SYSTEM PubSubTest
  (* Version 1.0, 2026-02-25, Administrateur *)
  APPLICATION PubSubTestApp
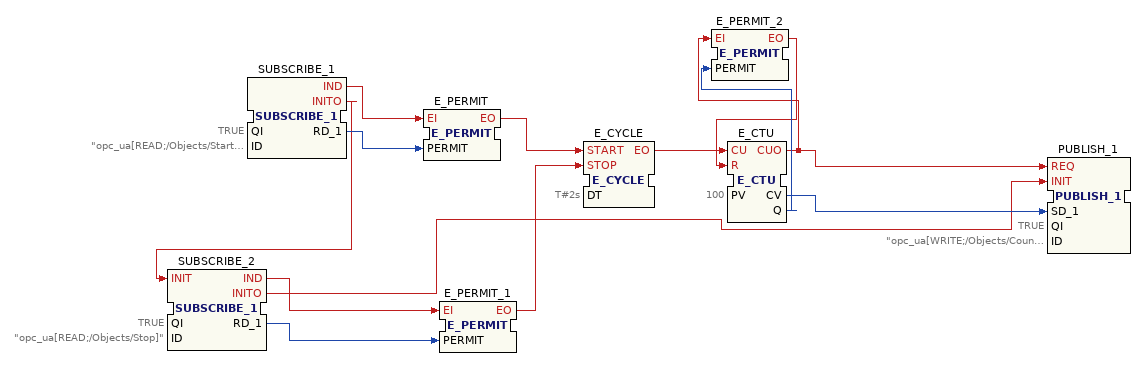
    FBS
      E_CYCLE : iec61499::events::E_CYCLE(DT := T#2s);
      E_CTU : iec61499::events::E_CTU(PV := 100);
      PUBLISH_1 : iec61499::net::PUBLISH_1(QI := TRUE, ID := "opc_ua[WRITE;/Objects/Counter]");
      SUBSCRIBE_1 : iec61499::net::SUBSCRIBE_1(QI := TRUE, ID := "opc_ua[READ;/Objects/Start]");
      E_PERMIT : iec61499::events::E_PERMIT;
      SUBSCRIBE_2 : iec61499::net::SUBSCRIBE_1(QI := TRUE, ID := "opc_ua[READ;/Objects/Stop]");
      E_PERMIT_1 : iec61499::events::E_PERMIT;
      E_PERMIT_2 : iec61499::events::E_PERMIT;
    END_FBS
    EVENT_CONNECTIONS
      E_CYCLE.EO TO E_CTU.CU;
      E_CTU.CUO TO PUBLISH_1.REQ;
      SUBSCRIBE_1.IND TO E_PERMIT.EI;
      E_PERMIT.EO TO E_CYCLE.START;
      E_PERMIT_1.EO TO E_CYCLE.STOP;
      SUBSCRIBE_2.IND TO E_PERMIT_1.EI;
      SUBSCRIBE_1.INITO TO SUBSCRIBE_2.INIT;
      SUBSCRIBE_2.INITO TO PUBLISH_1.INIT;
      E_CTU.CUO TO E_PERMIT_2.EI;
      E_PERMIT_2.EO TO E_CTU.R;
    END_CONNECTIONS
    DATA_CONNECTIONS
      E_CTU.CV TO PUBLISH_1.SD_1;
      SUBSCRIBE_1.RD_1 TO E_PERMIT.PERMIT;
      SUBSCRIBE_2.RD_1 TO E_PERMIT_1.PERMIT;
      E_CTU.Q TO E_PERMIT_2.PERMIT;
    END_CONNECTIONS
  END_APPLICATION
  DEVICE FORTE_PC : iec61499::system::FORTE_PC(MGR_ID := "localhost:61499" (* Device manager socket ID *))
    {SET_ATTRIBUTE(Profile, HOLOBLOC)}
    RESOURCE EMB_RES : iec61499::system::EMB_RES
      EVENT_CONNECTIONS
        START.WARM TO PubSubTestApp.SUBSCRIBE_1.INIT;
        START.COLD TO PubSubTestApp.SUBSCRIBE_1.INIT;
      END_CONNECTIONS
    END_RESOURCE
  END_DEVICE
  MAPPINGS
    PubSubTestApp.E_CYCLE ON FORTE_PC.EMB_RES;
    PubSubTestApp.E_CTU ON FORTE_PC.EMB_RES;
    PubSubTestApp.PUBLISH_1 ON FORTE_PC.EMB_RES;
    PubSubTestApp.E_PERMIT ON FORTE_PC.EMB_RES;
    PubSubTestApp.SUBSCRIBE_1 ON FORTE_PC.EMB_RES;
    PubSubTestApp.SUBSCRIBE_2 ON FORTE_PC.EMB_RES;
    PubSubTestApp.E_PERMIT_1 ON FORTE_PC.EMB_RES;
    PubSubTestApp.E_PERMIT_2 ON FORTE_PC.EMB_RES;
  END_MAPPINGS
  SEGMENTS
    Ethernet : iec61499::system::Ethernet;
  END_SEGMENTS
  LINKS
    FORTE_PC => Ethernet;
  END_LINKS
END_SYSTEM
